% RSLogix 500 project P4 - Multiposition Servo App v1.RSS, saved by version 8.30.00.16 %
PROJECT "PROJECT4"    % processor: Bul.1763 MicroLogix 1100 Series B %

PROGRAM FILES
  LAD 2 "MAIN"  3 rungs
  LAD 3 "I/O"  7 rungs
  LAD 4 "CONTROL"  9 rungs
  LAD 5 "CYCLE CALL"  23 rungs
  LAD 6 "TRAVELLING"  9 rungs

DATA FILES
  O0 OUTPUT  4 elements
  I1 INPUT  6 elements
  S2 STATUS  66 elements
  B3 BINARY  4 elements
  T4 TIMER  9 elements
  C5 COUNTER  1 elements
  R6 CONTROL  1 elements
  N7 INTEGER  2 elements
  F8 FLOAT  1 elements

LADDER 2 "MAIN"
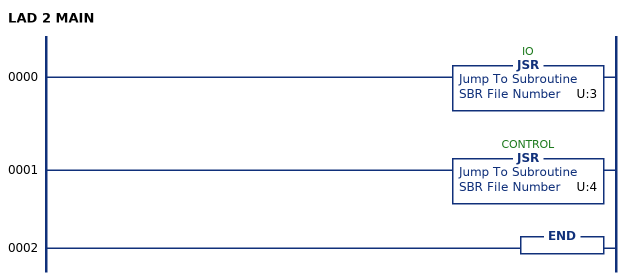
% Rung: 0 %
SOR JSR U:3 EOR
%   U:3  "IO" %
% Rung: 1 %
SOR JSR U:4 EOR
%   U:4  "CONTROL" %
% Rung: 2 %
SOR END EOR

LADDER 3 "I/O"
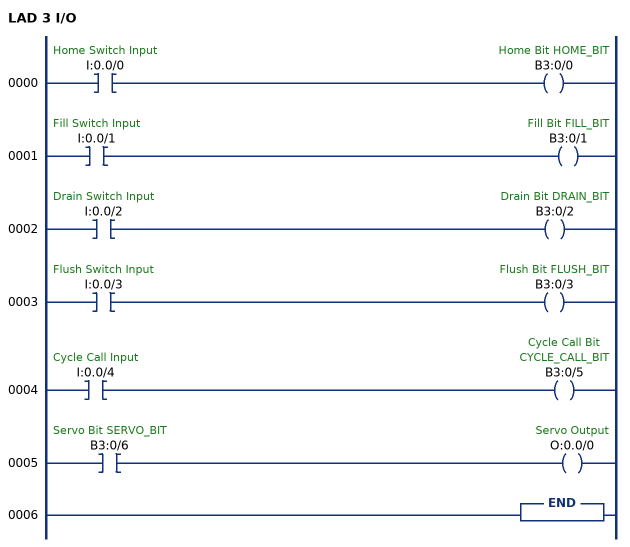
% Rung: 0 %
SOR XIC I:0.0/0 OTE B3:0/0 EOR
%   I:0.0/0  "Home Switch Input" %
%   B3:0/0  HOME_BIT  "Home Bit" %
% Rung: 1 %
SOR XIC I:0.0/1 OTE B3:0/1 EOR
%   I:0.0/1  "Fill Switch Input" %
%   B3:0/1  FILL_BIT  "Fill Bit" %
% Rung: 2 %
SOR XIC I:0.0/2 OTE B3:0/2 EOR
%   I:0.0/2  "Drain Switch Input" %
%   B3:0/2  DRAIN_BIT  "Drain Bit" %
% Rung: 3 %
SOR XIC I:0.0/3 OTE B3:0/3 EOR
%   I:0.0/3  "Flush Switch Input" %
%   B3:0/3  FLUSH_BIT  "Flush Bit" %
% Rung: 4 %
SOR XIC I:0.0/4 OTE B3:0/5 EOR
%   I:0.0/4  "Cycle Call Input" %
%   B3:0/5  CYCLE_CALL_BIT  "Cycle Call Bit" %
% Rung: 5 %
SOR XIC B3:0/6 OTE O:0.0/0 EOR
%   B3:0/6  SERVO_BIT  "Servo Bit" %
%   O:0.0/0  "Servo Output" %
% Rung: 6 %
SOR END EOR

LADDER 4 "CONTROL"
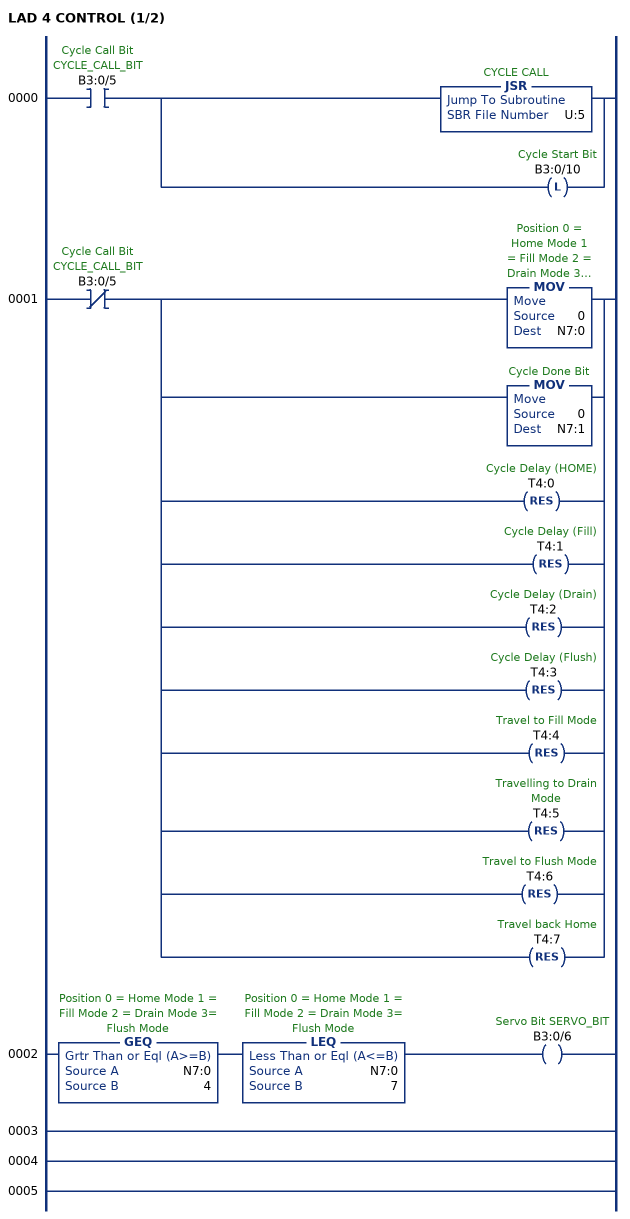
% Rung: 0 %
SOR XIC B3:0/5 BST JSR U:5 NXB OTL B3:0/10 BND EOR
%   B3:0/5  CYCLE_CALL_BIT  "Cycle Call Bit" %
%   U:5  "CYCLE CALL" %
%   B3:0/10  "Cycle Start Bit" %
% Rung: 1 %
SOR XIO B3:0/5 BST MOV 0 N7:0 NXB MOV 0 N7:1 NXB RES T4:0 NXB RES T4:1 NXB RES T4:2 NXB RES T4:3 NXB RES T4:4 NXB RES T4:5 NXB RES T4:6 NXB RES T4:7 BND EOR
%   B3:0/5  CYCLE_CALL_BIT  "Cycle Call Bit" %
%   N7:0  "Position 0 = Home Mode 1 = Fill Mode 2 = Drain Mode 3= Flush Mode" %
%   N7:1  "Cycle Done Bit" %
%   T4:0  "Cycle Delay (HOME)" %
%   T4:1  "Cycle Delay (Fill)" %
%   T4:2  "Cycle Delay (Drain)" %
%   T4:3  "Cycle Delay (Flush)" %
%   T4:4  "Travel to Fill Mode" %
%   T4:5  "Travelling to Drain Mode" %
%   T4:6  "Travel to Flush Mode" %
%   T4:7  "Travel back Home" %
% Rung: 2 %
SOR GEQ N7:0 4 LEQ N7:0 7 OTE B3:0/6 EOR
%   N7:0  "Position 0 = Home Mode 1 = Fill Mode 2 = Drain Mode 3= Flush Mode" %
%   B3:0/6  SERVO_BIT  "Servo Bit" %
% Rung: 3 %  % edit flag set %
SOR EOR
% Rung: 4 %  % edit flag set %
SOR EOR
% Rung: 5 %  % edit flag set %
SOR EOR

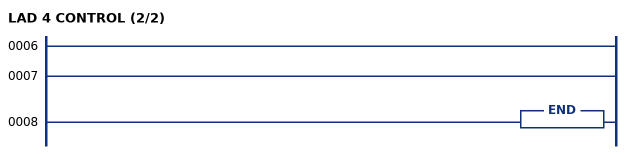
% Rung: 6 %  % edit flag set %
SOR EOR
% Rung: 7 %  % edit flag set %
SOR EOR
% Rung: 8 %
SOR END EOR

LADDER 5 "CYCLE CALL"
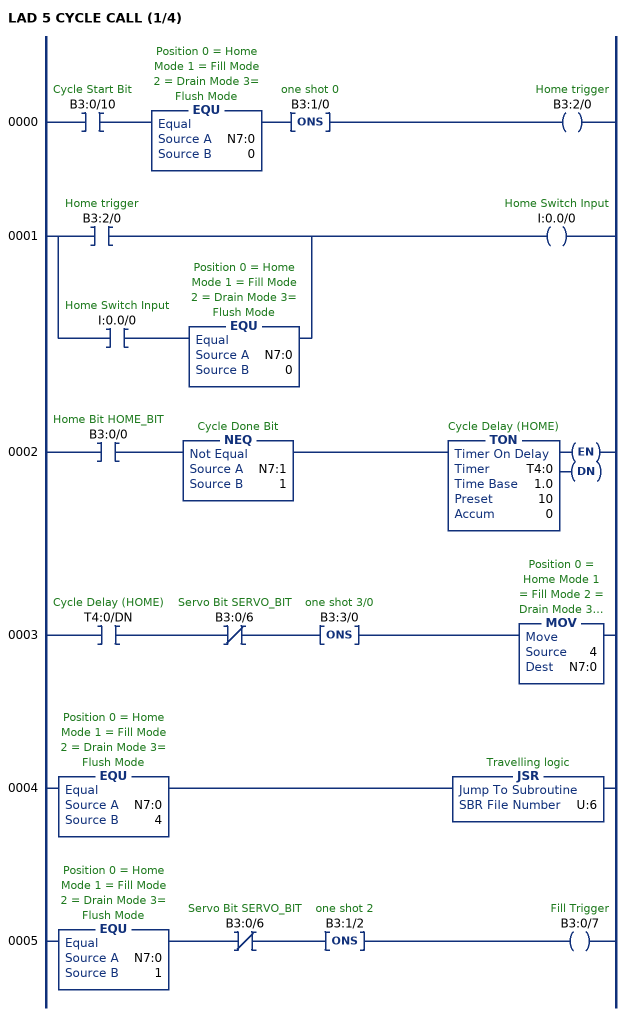
% Rung: 0 %
SOR XIC B3:0/10 EQU N7:0 0 ONS B3:1/0 OTE B3:2/0 EOR
%   B3:0/10  "Cycle Start Bit" %
%   N7:0  "Position 0 = Home Mode 1 = Fill Mode 2 = Drain Mode 3= Flush Mode" %
%   B3:1/0  "one shot 0" %
%   B3:2/0  "Home trigger" %
% Rung: 1 %
SOR BST XIC B3:2/0 NXB XIC I:0.0/0 EQU N7:0 0 BND OTE I:0.0/0 EOR
%   B3:2/0  "Home trigger" %
%   I:0.0/0  "Home Switch Input" %
%   N7:0  "Position 0 = Home Mode 1 = Fill Mode 2 = Drain Mode 3= Flush Mode" %
% Rung: 2 %
SOR XIC B3:0/0 NEQ N7:1 1 TON T4:0 1.0 10 0 EOR
%   B3:0/0  HOME_BIT  "Home Bit" %
%   N7:1  "Cycle Done Bit" %
%   T4:0  "Cycle Delay (HOME)" %
% Rung: 3 %
SOR XIC T4:0/DN XIO B3:0/6 ONS B3:3/0 MOV 4 N7:0 EOR
%   T4:0  "Cycle Delay (HOME)" %
%   B3:0/6  SERVO_BIT  "Servo Bit" %
%   B3:3/0  "one shot 3/0" %
%   N7:0  "Position 0 = Home Mode 1 = Fill Mode 2 = Drain Mode 3= Flush Mode" %
% Rung: 4 %
SOR EQU N7:0 4 JSR U:6 EOR
%   N7:0  "Position 0 = Home Mode 1 = Fill Mode 2 = Drain Mode 3= Flush Mode" %
%   U:6  "Travelling logic" %
% Rung: 5 %
SOR EQU N7:0 1 XIO B3:0/6 ONS B3:1/2 OTE B3:0/7 EOR
%   N7:0  "Position 0 = Home Mode 1 = Fill Mode 2 = Drain Mode 3= Flush Mode" %
%   B3:0/6  SERVO_BIT  "Servo Bit" %
%   B3:1/2  "one shot 2" %
%   B3:0/7  "Fill Trigger" %

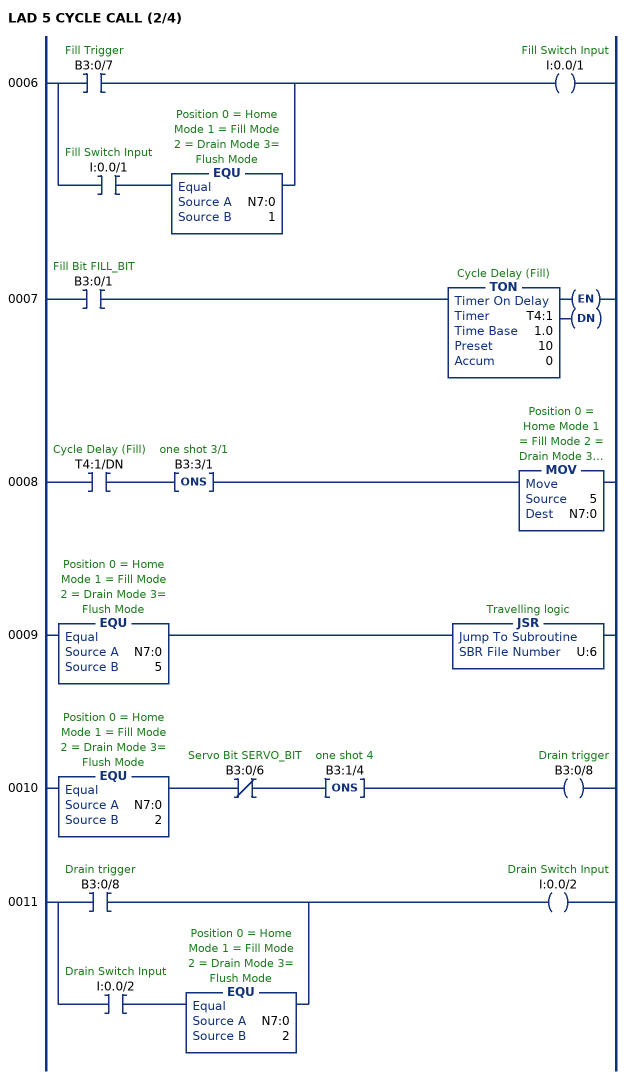
% Rung: 6 %
SOR BST XIC B3:0/7 NXB XIC I:0.0/1 EQU N7:0 1 BND OTE I:0.0/1 EOR
%   B3:0/7  "Fill Trigger" %
%   I:0.0/1  "Fill Switch Input" %
%   N7:0  "Position 0 = Home Mode 1 = Fill Mode 2 = Drain Mode 3= Flush Mode" %
% Rung: 7 %
SOR XIC B3:0/1 TON T4:1 1.0 10 0 EOR
%   B3:0/1  FILL_BIT  "Fill Bit" %
%   T4:1  "Cycle Delay (Fill)" %
% Rung: 8 %
SOR XIC T4:1/DN ONS B3:3/1 MOV 5 N7:0 EOR
%   T4:1  "Cycle Delay (Fill)" %
%   B3:3/1  "one shot 3/1" %
%   N7:0  "Position 0 = Home Mode 1 = Fill Mode 2 = Drain Mode 3= Flush Mode" %
% Rung: 9 %
SOR EQU N7:0 5 JSR U:6 EOR
%   N7:0  "Position 0 = Home Mode 1 = Fill Mode 2 = Drain Mode 3= Flush Mode" %
%   U:6  "Travelling logic" %
% Rung: 10 %
SOR EQU N7:0 2 XIO B3:0/6 ONS B3:1/4 OTE B3:0/8 EOR
%   N7:0  "Position 0 = Home Mode 1 = Fill Mode 2 = Drain Mode 3= Flush Mode" %
%   B3:0/6  SERVO_BIT  "Servo Bit" %
%   B3:1/4  "one shot 4" %
%   B3:0/8  "Drain trigger" %
% Rung: 11 %
SOR BST XIC B3:0/8 NXB XIC I:0.0/2 EQU N7:0 2 BND OTE I:0.0/2 EOR
%   B3:0/8  "Drain trigger" %
%   I:0.0/2  "Drain Switch Input" %
%   N7:0  "Position 0 = Home Mode 1 = Fill Mode 2 = Drain Mode 3= Flush Mode" %

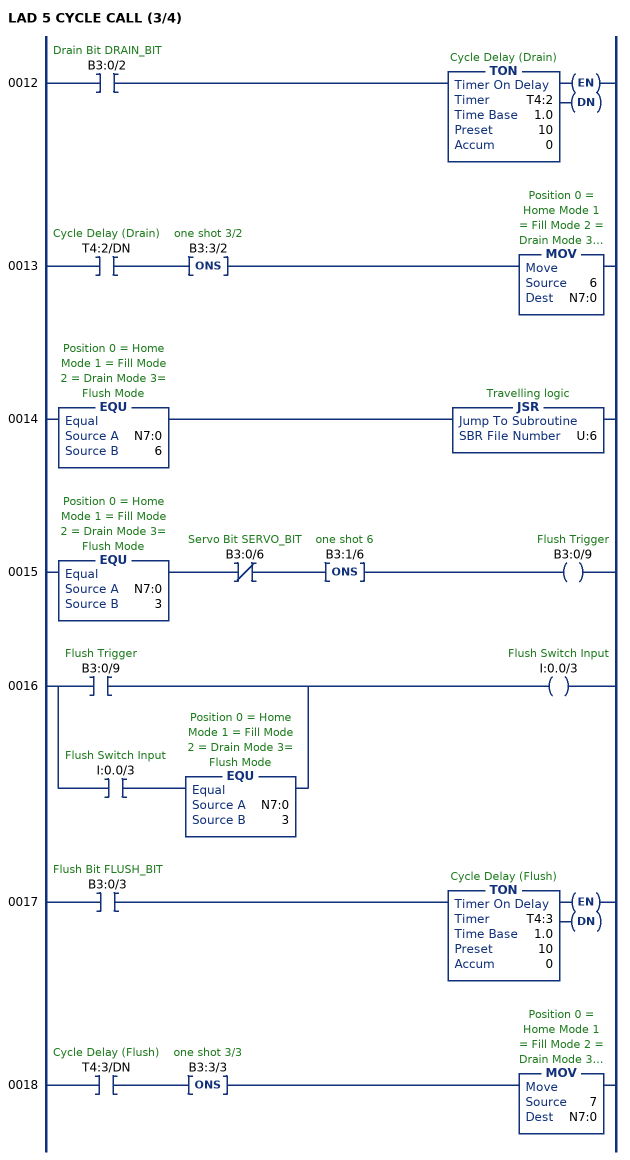
% Rung: 12 %
SOR XIC B3:0/2 TON T4:2 1.0 10 0 EOR
%   B3:0/2  DRAIN_BIT  "Drain Bit" %
%   T4:2  "Cycle Delay (Drain)" %
% Rung: 13 %
SOR XIC T4:2/DN ONS B3:3/2 MOV 6 N7:0 EOR
%   T4:2  "Cycle Delay (Drain)" %
%   B3:3/2  "one shot 3/2" %
%   N7:0  "Position 0 = Home Mode 1 = Fill Mode 2 = Drain Mode 3= Flush Mode" %
% Rung: 14 %
SOR EQU N7:0 6 JSR U:6 EOR
%   N7:0  "Position 0 = Home Mode 1 = Fill Mode 2 = Drain Mode 3= Flush Mode" %
%   U:6  "Travelling logic" %
% Rung: 15 %
SOR EQU N7:0 3 XIO B3:0/6 ONS B3:1/6 OTE B3:0/9 EOR
%   N7:0  "Position 0 = Home Mode 1 = Fill Mode 2 = Drain Mode 3= Flush Mode" %
%   B3:0/6  SERVO_BIT  "Servo Bit" %
%   B3:1/6  "one shot 6" %
%   B3:0/9  "Flush Trigger" %
% Rung: 16 %
SOR BST XIC B3:0/9 NXB XIC I:0.0/3 EQU N7:0 3 BND OTE I:0.0/3 EOR
%   B3:0/9  "Flush Trigger" %
%   I:0.0/3  "Flush Switch Input" %
%   N7:0  "Position 0 = Home Mode 1 = Fill Mode 2 = Drain Mode 3= Flush Mode" %
% Rung: 17 %
SOR XIC B3:0/3 TON T4:3 1.0 10 0 EOR
%   B3:0/3  FLUSH_BIT  "Flush Bit" %
%   T4:3  "Cycle Delay (Flush)" %
% Rung: 18 %
SOR XIC T4:3/DN ONS B3:3/3 MOV 7 N7:0 EOR
%   T4:3  "Cycle Delay (Flush)" %
%   B3:3/3  "one shot 3/3" %
%   N7:0  "Position 0 = Home Mode 1 = Fill Mode 2 = Drain Mode 3= Flush Mode" %

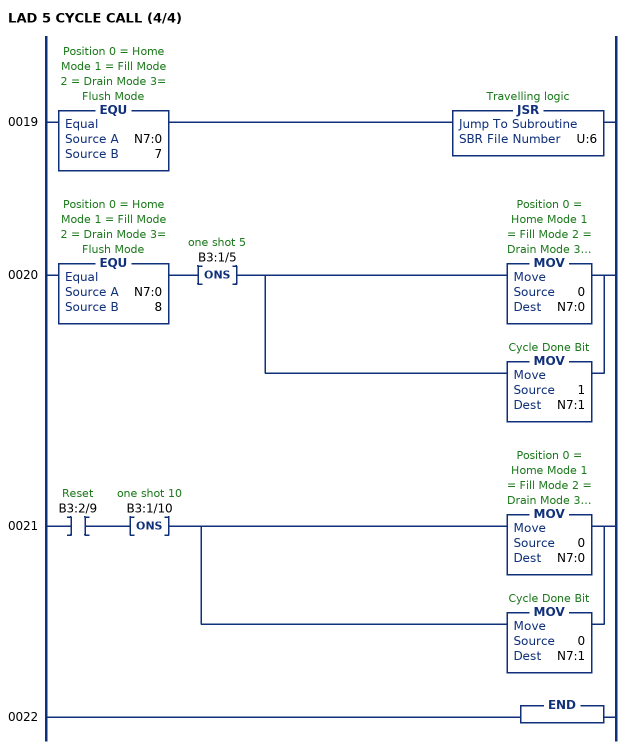
% Rung: 19 %
SOR EQU N7:0 7 JSR U:6 EOR
%   N7:0  "Position 0 = Home Mode 1 = Fill Mode 2 = Drain Mode 3= Flush Mode" %
%   U:6  "Travelling logic" %
% Rung: 20 %
SOR EQU N7:0 8 ONS B3:1/5 BST MOV 0 N7:0 NXB MOV 1 N7:1 BND EOR
%   N7:0  "Position 0 = Home Mode 1 = Fill Mode 2 = Drain Mode 3= Flush Mode" %
%   B3:1/5  "one shot 5" %
%   N7:1  "Cycle Done Bit" %
% Rung: 21 %
SOR XIC B3:2/9 ONS B3:1/10 BST MOV 0 N7:0 NXB MOV 0 N7:1 BND EOR
%   B3:2/9  "Reset" %
%   B3:1/10  "one shot 10" %
%   N7:0  "Position 0 = Home Mode 1 = Fill Mode 2 = Drain Mode 3= Flush Mode" %
%   N7:1  "Cycle Done Bit" %
% Rung: 22 %
SOR END EOR

LADDER 6 "TRAVELLING"
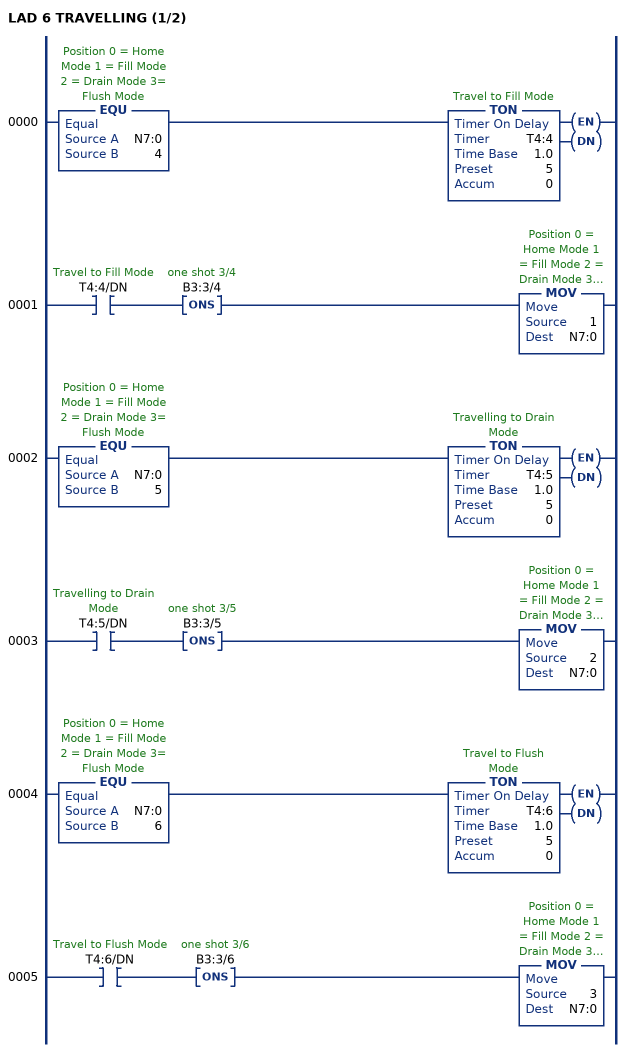
% Rung: 0 %
SOR EQU N7:0 4 TON T4:4 1.0 5 0 EOR
%   N7:0  "Position 0 = Home Mode 1 = Fill Mode 2 = Drain Mode 3= Flush Mode" %
%   T4:4  "Travel to Fill Mode" %
% Rung: 1 %
SOR XIC T4:4/DN ONS B3:3/4 MOV 1 N7:0 EOR
%   T4:4  "Travel to Fill Mode" %
%   B3:3/4  "one shot 3/4" %
%   N7:0  "Position 0 = Home Mode 1 = Fill Mode 2 = Drain Mode 3= Flush Mode" %
% Rung: 2 %
SOR EQU N7:0 5 TON T4:5 1.0 5 0 EOR
%   N7:0  "Position 0 = Home Mode 1 = Fill Mode 2 = Drain Mode 3= Flush Mode" %
%   T4:5  "Travelling to Drain Mode" %
% Rung: 3 %
SOR XIC T4:5/DN ONS B3:3/5 MOV 2 N7:0 EOR
%   T4:5  "Travelling to Drain Mode" %
%   B3:3/5  "one shot 3/5" %
%   N7:0  "Position 0 = Home Mode 1 = Fill Mode 2 = Drain Mode 3= Flush Mode" %
% Rung: 4 %
SOR EQU N7:0 6 TON T4:6 1.0 5 0 EOR
%   N7:0  "Position 0 = Home Mode 1 = Fill Mode 2 = Drain Mode 3= Flush Mode" %
%   T4:6  "Travel to Flush Mode" %
% Rung: 5 %
SOR XIC T4:6/DN ONS B3:3/6 MOV 3 N7:0 EOR
%   T4:6  "Travel to Flush Mode" %
%   B3:3/6  "one shot 3/6" %
%   N7:0  "Position 0 = Home Mode 1 = Fill Mode 2 = Drain Mode 3= Flush Mode" %

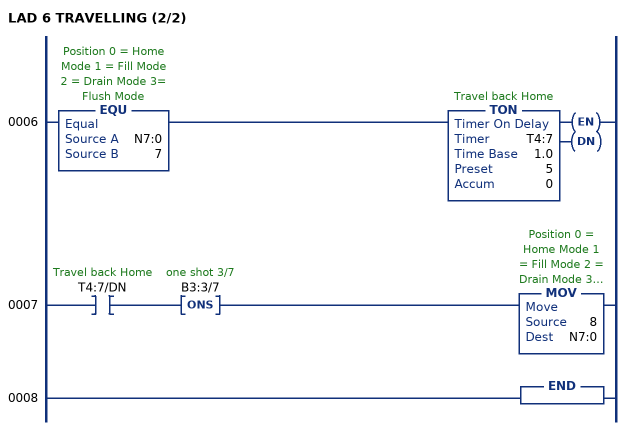
% Rung: 6 %
SOR EQU N7:0 7 TON T4:7 1.0 5 0 EOR
%   N7:0  "Position 0 = Home Mode 1 = Fill Mode 2 = Drain Mode 3= Flush Mode" %
%   T4:7  "Travel back Home" %
% Rung: 7 %
SOR XIC T4:7/DN ONS B3:3/7 MOV 8 N7:0 EOR
%   T4:7  "Travel back Home" %
%   B3:3/7  "one shot 3/7" %
%   N7:0  "Position 0 = Home Mode 1 = Fill Mode 2 = Drain Mode 3= Flush Mode" %
% Rung: 8 %
SOR END EOR

OTHER DOCUMENTED ADDRESSES
  B3:0/4  "TRAVELLING Bit"
  B3:0/11  "one shot 11"
  B3:0/12  "CYCLE DONE BIT"
  B3:1/1  "one shot 1"
  B3:1/3  "one shot 3"
  B3:1/7  "one shot 7"
  B3:1/8  "one shot 8"
  B3:1/9  "one shot 9"
  B3:1/11  "One shot 11"
  B3:2/1  "Fill Trigger"
  B3:2/2  "Drain Trigger"
  B3:2/3  "Home-Fill bit"
  B3:2/4  "Fill-Drain Bit"
  B3:2/5  "Drain-Flush Bit"
  B3:2/6  "Flush-Home Bit"
  B3:2/7  "Trigger"
  B3:2/8  "Inturrupt"
  T4:8  "Restart Delay"

DATA TABLE (non-zero values as saved)
DATA T4
% .PRE .ACC %
% T4:0 % 10 0
% T4:1 % 10 0
% T4:2 % 10 0
% T4:3 % 10 0
% T4:4 % 5 0
% T4:5 % 5 0
% T4:6 % 5 0
% T4:7 % 5 0
% T4:8 % 5 0
DATA N7
% N7:0 % 8 0
